// TIA Portal V20 export
DATA_BLOCK "PM3"   // DB277
// stored: MemoryReserve 100
   VAR
      "TOP TAPE CUTTER UP" : Bool;
      "TOP TAPE CUTTER DOWN" : Bool;
      "TOP TAPE CUTTER CLAMP UP" : Bool;
      "TOP TAPE CUTTER CLAMP DOWN" : Bool;
      "TOP TAPE CLAMP OPEN" : Bool;
      "TOP TAPE CLAMP CLOSE" : Bool;
      "TOP TAPE TENSION FORWARD" : Bool;
      "TOP TAPE TENSION BACKWARD" : Bool;
      "TOP TAPE LOADING FORWARD" : Bool;
      "TOP TAPE LOADING BACKWARD" : Bool;
      "TOP TAPE ATTACHMENT UP" : Bool;
      "TOP TAPE ATTACHMENT DOWN" : Bool;
      SPARE : Bool;
      SPARE_1 : Bool;
      SPARE_2 : Bool;
      SPARE_3 : Bool;
   END_VAR
BEGIN
END_DATA_BLOCK
